// TIA Portal V18 export
VAR_GLOBAL   // PLC tag table "DO"
   "H/SSR_006_XV01_OPEN" AT %Q0.0 : Bool;
   "H/SSR_006_XV02_OPEN" AT %Q0.1 : Bool;
   "H/SSR_006_XV03_OPEN" AT %Q0.2 : Bool;
   "H/SSR_006_XV04_OPEN" AT %Q0.3 : Bool;
   "H/SSR_006_XV05_OPEN" AT %Q0.4 : Bool;
   "H/SSR_006_XV06_OPEN" AT %Q0.5 : Bool;
   "H/SSR_006_XV07_OPEN" AT %Q0.6 : Bool;
   "H/SSR_006_XV08_OPEN" AT %Q0.7 : Bool;
   "H/SSR_006_XV09_OPEN" AT %Q1.0 : Bool;
   "H/SSR_006_XV10_OPEN" AT %Q1.1 : Bool;
   "H/SSR_006_XV11_OPEN" AT %Q1.2 : Bool;
   "H/SSR_006_XV12_OPEN" AT %Q1.3 : Bool;
   "H/SSR_006_XV13_OPEN" AT %Q1.4 : Bool;
   "H/SSR_006_XV14_OPEN" AT %Q1.5 : Bool;
   "H/SSR_006_AG_RUN" AT %Q1.6 : Bool;
   "H/SSR_010_XV01_OPEN" AT %Q1.7 : Bool;
   "H/SSR_010_XV02_OPEN" AT %Q2.0 : Bool;
   "H/SSR_010_XV03_OPEN" AT %Q2.1 : Bool;
   "H/SSR_010_XV04_OPEN" AT %Q2.2 : Bool;
   "H/SSR_010_XV05_OPEN" AT %Q2.3 : Bool;
   "H/SSR_010_XV06_OPEN" AT %Q2.4 : Bool;
   "H/SSR_010_XV07_OPEN" AT %Q2.5 : Bool;
   "H/SSR_010_XV08_OPEN" AT %Q2.6 : Bool;
   "H/SSR_010_XV09_OPEN" AT %Q2.7 : Bool;
   "H/SSR_010_XV10_OPEN" AT %Q3.0 : Bool;
   "H/SSR_010_XV11_OPEN" AT %Q3.1 : Bool;
   "H/SSR_010_XV12_OPEN" AT %Q3.2 : Bool;
   "H/SSR_010_XV13_OPEN" AT %Q3.3 : Bool;
   "H/SSR_010_XV14_OPEN" AT %Q3.4 : Bool;
   "H/SSR_010_AG_RUN" AT %Q3.5 : Bool;
   "H/SSR_019_XV01_OPEN" AT %Q3.6 : Bool;
   "H/SSR_019_XV02_OPEN" AT %Q3.7 : Bool;
   "H/SSR_019_XV03_OPEN" AT %Q4.0 : Bool;
   "H/SSR_019_XV04_OPEN" AT %Q4.1 : Bool;
   "H/SSR_019_XV05_OPEN" AT %Q4.2 : Bool;
   "H/SSR_019_XV06_OPEN" AT %Q4.3 : Bool;
   "H/SSR_019_XV07_OPEN" AT %Q4.4 : Bool;
   "H/SSR_019_XV08_OPEN" AT %Q4.5 : Bool;
   "H/SSR_019_XV09_OPEN" AT %Q4.6 : Bool;
   "H/SSR_019_XV10_OPEN" AT %Q4.7 : Bool;
   "H/SSR_019_XV11_OPEN" AT %Q5.0 : Bool;
   "H/SSR_019_XV12_OPEN" AT %Q5.1 : Bool;
   "H/SSR_019_XV13_OPEN" AT %Q5.2 : Bool;
   "H/SSR_019_XV14_OPEN" AT %Q5.3 : Bool;
   "H/SSR_019_AG_RUN" AT %Q5.4 : Bool;
   "H/SSR_020_XV01_OPEN" AT %Q5.5 : Bool;
   "H/SSR_020_XV02_OPEN" AT %Q5.6 : Bool;
   "H/SSR_020_XV03_OPEN" AT %Q5.7 : Bool;
   "H/SSR_020_XV04_OPEN" AT %Q6.0 : Bool;
   "H/SSR_020_XV05_OPEN" AT %Q6.1 : Bool;
   "H/SSR_020_XV06_OPEN" AT %Q6.2 : Bool;
   "H/SSR_020_XV07_OPEN" AT %Q6.3 : Bool;
   "H/SSR_020_XV08_OPEN" AT %Q6.4 : Bool;
   "H/SSR_020_XV09_OPEN" AT %Q6.5 : Bool;
   "H/SSR_020_XV10_OPEN" AT %Q6.6 : Bool;
   "H/SSR_020_XV11_OPEN" AT %Q6.7 : Bool;
   "H/SSR_020_XV12_OPEN" AT %Q7.0 : Bool;
   "H/SSR_020_XV13_OPEN" AT %Q7.1 : Bool;
   "H/SSR_020_XV14_OPEN" AT %Q7.2 : Bool;
   "H/SSR_020_AG_RUN" AT %Q7.3 : Bool;
   DO_SPARE_1 AT %Q7.4 : Bool;
   DO_SPARE_2 AT %Q7.5 : Bool;
   DO_SPARE_3 AT %Q7.6 : Bool;
   DO_SPARE_4 AT %Q7.7 : Bool;
   DO_SPARE_5 AT %Q8.0 : Bool;
   DO_SPARE_6 AT %Q8.1 : Bool;
   DO_SPARE_7 AT %Q8.2 : Bool;
   DO_SPARE_8 AT %Q8.3 : Bool;
   DO_SPARE_9 AT %Q8.4 : Bool;
   DO_SPARE_10 AT %Q8.5 : Bool;
   DO_SPARE_11 AT %Q8.6 : Bool;
   DO_SPARE_12 AT %Q8.7 : Bool;
   DO_SPARE_13 AT %Q9.0 : Bool;
   DO_SPARE_14 AT %Q9.1 : Bool;
   DO_SPARE_15 AT %Q9.2 : Bool;
   DO_SPARE_16 AT %Q9.3 : Bool;
   DO_SPARE_17 AT %Q9.4 : Bool;
   DO_SPARE_18 AT %Q9.5 : Bool;
   DO_SPARE_19 AT %Q9.6 : Bool;
   DO_SPARE_20 AT %Q9.7 : Bool;
   DO_SPARE_21 AT %Q10.0 : Bool;
   DO_SPARE_22 AT %Q10.1 : Bool;
   DO_SPARE_23 AT %Q10.2 : Bool;
   DO_SPARE_24 AT %Q10.3 : Bool;
   DO_SPARE_25 AT %Q10.4 : Bool;
   DO_SPARE_26 AT %Q10.5 : Bool;
   DO_SPARE_27 AT %Q10.6 : Bool;
   DO_SPARE_28 AT %Q10.7 : Bool;
   DO_SPARE_29 AT %Q11.0 : Bool;
   DO_SPARE_30 AT %Q11.1 : Bool;
   DO_SPARE_31 AT %Q11.2 : Bool;
   DO_SPARE_32 AT %Q11.3 : Bool;
   DO_SPARE_33 AT %Q11.4 : Bool;
   DO_SPARE_34 AT %Q11.5 : Bool;
   DO_SPARE_35 AT %Q11.6 : Bool;
   DO_SPARE_36 AT %Q11.7 : Bool;
   DO_SPARE_37 AT %Q12.0 : Bool;
   DO_SPARE_38 AT %Q12.1 : Bool;
   DO_SPARE_39 AT %Q12.2 : Bool;
   DO_SPARE_40 AT %Q12.3 : Bool;
   DO_SPARE_41 AT %Q12.4 : Bool;
   DO_SPARE_42 AT %Q12.5 : Bool;
   DO_SPARE_43 AT %Q12.6 : Bool;
   DO_SPARE_44 AT %Q12.7 : Bool;
   DO_SPARE_45 AT %Q13.0 : Bool;
   DO_SPARE_46 AT %Q13.1 : Bool;
   DO_SPARE_47 AT %Q13.2 : Bool;
   DO_SPARE_48 AT %Q13.3 : Bool;
   DO_SPARE_49 AT %Q13.4 : Bool;
   DO_SPARE_50 AT %Q13.5 : Bool;
   DO_SPARE_51 AT %Q13.6 : Bool;
   DO_SPARE_52 AT %Q13.7 : Bool;
END_VAR
